INTERFACE I_TagAssignment

METHOD AA1 : BOOL
VAR_INPUT
END_VAR
END_METHOD

METHOD AA2 : BOOL
VAR_INPUT
END_VAR
END_METHOD

METHOD DCM : BOOL
VAR_INPUT
END_VAR
END_METHOD

METHOD MVA : BOOL
VAR_INPUT
END_VAR
END_METHOD

METHOD MVB : BOOL
VAR_INPUT
END_VAR
END_METHOD

METHOD R1 : BOOL
VAR_INPUT
END_VAR
END_METHOD

METHOD R2 : BOOL
VAR_INPUT
END_VAR
END_METHOD

METHOD R3 : BOOL
VAR_INPUT
END_VAR
END_METHOD

METHOD R4 : BOOL
VAR_INPUT
END_VAR
END_METHOD

METHOD R5 : BOOL
VAR_INPUT
END_VAR
END_METHOD

METHOD RV : BOOL
VAR_INPUT
END_VAR
END_METHOD

END_INTERFACE

(* stored: Version 1.1.0.1, ProductVersion 3.1.4024.6
   Itf I_TagAssignment: Id {2dface39-54e7-4a27-85ee-612eb6543226}
   Method AA1: Id {ca9802ad-c522-4e6c-a620-c230b2bcbd89}
   Method AA2: Id {40d73585-59d1-40d6-a6a9-b8b1fabe94be}
   Method DCM: Id {cbd7a888-8f42-4ec5-98a4-1ebc65f6ae46}
   Method MVA: Id {c91a9a6f-4cca-4baa-b620-10d1934acfec}
   Method MVB: Id {c2bf5e29-92d3-477a-b64f-9b10287a1589}
   Method R1: Id {64014a1e-2d2b-4be0-a505-8dd25b6a4924}
   Method R2: Id {8c4e5655-d103-498e-b21c-aeef081ab15c}
   Method R3: Id {03156c94-07f6-4609-85b2-4f32791f9075}
   Method R4: Id {831b4d41-c642-473b-a36f-142647e79b20}
   Method R5: Id {248eba15-7dd6-47ac-a0e8-1cda66179fe7}
   Method RV: Id {d1dfa7b8-a737-4382-9552-c2b263406157} *)
